//Request var
	eRequestedProfile		: E_AXIS_MOVE_PROFILE := E_AXIS_MOVE_PROFILE.Slow;
	rRequestedTarget		: LREAL := 0;
	Profile				    	: ARRAY[0..2]OF ST_AXIS_MOVE_PROFILE ;
END_VAR

IF NOT bInit THEN
  RETURN;
END_IF

//CALL BLOCK
fbPower(Axis:= _AxisREF_P^, Override:= lrAxisOverride);
fbStop(Axis:= _AxisREF_P^);
fbReset(Axis:= _AxisREF_P^);
fbHome( Axis:= _AxisREF_P^, bCalibrationCam:=_udCalibrationSensor_P^.19,
		    Options := stHomingOption, Position := lrnOffsetExtractorHoming);
fbHomeInv( Axis:= _AxisREF_P^, bCalibrationCam:=_udCalibrationSensor_P^.19,
		    Options := stHomingInvOption, Position := lrnOffsetExtractorHoming);
fbMoveAbso(Axis:= _AxisREF_P^);
fbReadStatus(Axis:= _AxisREF_P^,Enable := TRUE);
fbMoveJog(Axis := _AxisREF_P^,JogForward := stJogControl.bMoveFW, JogBackwards := stJogControl.bMoveBW);
fbTimeRetryHomming(IN := nStep = E_StepAxis.AbortHoming);
fbTimeAbortHoming(IN := nStep = E_StepAxis.RetryHoming);
fbTimeOutReset(IN := nStep = E_StepAxis.InitReset);
fbTrigErrorMotor(CLK := _AxisREF_P^.NcToPlc.ErrorCode <> 0);
_lrActPos := _AxisREF_P^.NcToPlc.ActPos;


IF fbTrigErrorMotor.Q THEN
  nStep := E_StepAxis.Idle;
  bRequestMoveAbso := FALSE;
  bRequestHoming := FALSE;
  fbHome.Execute := FALSE;
  fbHomeInv.Execute := FALSE;
  fbMoveAbso.Execute := FALSE;
END_IF

//Defect
objMotorError();
objMotorError.Set(bSetActivate := _AxisREF_P^.NcToPlc.ErrorCode <> 0 AND _AxisREF_P^.NcToPlc.ErrorCode <> 18000 );

objMoveAbsError();
objMoveAbsError.Set(bSetActivate := fbMoveAbso.Error AND fbMoveAbso.Execute);

objMotorResetError();
objMotorResetError.Set(bSetActivate := fbReset.Error AND fbReset.Execute);

//objMotorPowerError();
//objMotorPowerError.SetState(bSetActivate := fbPower.Error AND fbPower.Enable);

objHommingError();

// If bEnableMove is down, do a stop automatically
//IF NOT bEnableMove THEN
//	bRequestStop		:= TRUE;
//	eRequestedProfile	:= E_AXIS_MOVE_PROFILE.Fast;
//END_IF


CASE nStep OF
	// ------------------------------------------------------------------
	E_StepAxis.IDLE :	
		bRequestStop	:= FALSE;			
    IF bRequestPowerOff THEN
      nStep := E_StepAxis.PoweringOff;
      bRequestPowerOff	:= FALSE;
    ELSIF bRequestPowerOn THEN
      nStep := E_StepAxis.PoweringOn;
      bRequestPowerOn		:= FALSE;
    ELSIF bRequestMoveAbso THEN
      nStep := E_StepAxis.InitMoveAbs;
      bRequestMoveAbso	:= FALSE;
    ELSIF bRequestHoming THEN
      bRequestHoming		:= FALSE;
			IF _udCalibrationSensor_P^.19 THEN
				nStep := E_StepAxis.InitRetryHoming;
			ELSE
				nStep := E_StepAxis.InitHoming;
			END_IF	
    ELSIF bRequestReset OR (_AxisREF_P^.NcToPlc.ErrorCode <> 0) THEN
			//added to support MDF extractor: homing in both direction		
			nStep := E_StepAxis.InitReset;
      bRequestReset		:= FALSE;
    END_IF
	
	// ******************************************************************
	// --- POWER ---
	// ******************************************************************
		// ------------------------------------------------------------------
		E_StepAxis.PoweringOff :
      fbPower.Enable := FALSE;
			objHommingError.Set(Activate:= FALSE);
      IF NOT fbPower.Status THEN
        _bIsDone	:= TRUE;
        _bIsBusy	:= FALSE;
        nStep := E_StepAxis.IDLE;
      ELSIF fbPower.Error THEN
        nErrorId := fbPower.ErrorID;
        nStep := E_StepAxis.ERROR;
      END_IF
			
		// ------------------------------------------------------------------
		E_StepAxis.PoweringOn :
      fbPower.Enable			:= TRUE;
      fbPower.Enable_Positive	:= TRUE;
      fbPower.Enable_Negative	:= TRUE;
      IF fbPower.Status THEN
        _bIsDone	:= TRUE;
        _bIsBusy	:= FALSE;
        nStep  := E_StepAxis.Idle;
      ELSIF fbPower.Error THEN
        fbPower.Enable			:= FALSE;
        fbPower.Enable_Positive	:= FALSE;
        fbPower.Enable_Negative	:= FALSE;
        _bIsBusy	:= FALSE;
        nStep  := E_StepAxis.Idle;      
      END_IF
			
	// ******************************************************************
	// --- ABSOLUTE ---
	// ******************************************************************
		// ------------------------------------------------------------------
		E_StepAxis.InitMoveAbs:
      fbMoveAbso.Position		:= rRequestedTarget;
      fbMoveAbso.Velocity		:= Profile[eRequestedProfile].Velo;
      fbMoveAbso.Acceleration	:= Profile[eRequestedProfile].Acc;
      fbMoveAbso.Deceleration	:= Profile[eRequestedProfile].Dec;
      fbMoveAbso.Jerk			:= Profile[eRequestedProfile].Jerk;
      fbMoveAbso.Execute			:= TRUE;
      IF fbMoveAbso.Busy THEN
         nStep := E_StepAxis.MoveAbs;
      END_IF
    
    // ------------------------------------------------------------------  
    E_StepAxis.MoveAbs:    
      IF fbMoveAbso.Done THEN
        nStep:= E_StepAxis.EndMoveAbs;
      ELSIF bRequestStop THEN
        fbMoveAbso.Execute := FALSE;
        nStep:= E_StepAxis.InitStop;
        bRequestStop := FALSE;
      ELSIF fbMoveAbso.Error THEN
        fbMoveAbso.Execute	:= false;
        _bIsBusy	:= FALSE;
        nStep     := E_StepAxis.Idle;
      END_IF
     
    // ------------------------------------------------------------------  
    E_StepAxis.EndMoveAbs: 
      _bIsDone	:= TRUE;
      _bIsBusy	:= FALSE;
      fbMoveAbso.Execute  := FALSE;
      nStep     := E_StepAxis.Idle;
						
	// ******************************************************************
	// --- STOP ---
	// ******************************************************************
		// ------------------------------------------------------------------
		E_StepAxis.InitStop :
			bRequestStop	:= FALSE;
      fbStop.Deceleration	:= Profile[eRequestedProfile].Dec;
      fbStop.Jerk			    := Profile[eRequestedProfile].Jerk;
      fbStop.Execute		  := TRUE;
      IF fbStop.Busy THEN
        nStep := E_StepAxis.Stopping;
			END_IF
                  
		// ------------------------------------------------------------------
		E_StepAxis.Stopping :        
      IF _AxisREF_P^.Status.NotMoving THEN
        _bIsDone	:= TRUE;
        _bIsBusy	:= FALSE;
        nStep  := E_StepAxis.EndStopping;
      END_IF
        
		// ------------------------------------------------------------------
		E_StepAxis.EndStopping :        
      fbStop.Execute	:= FALSE;
      objHommingError.Set(Activate:= FALSE);
			nStep           := E_StepAxis.Idle;

	// ******************************************************************
	// --- HOMING ---
	// ******************************************************************
		// ------------------------------------------------------------------
		E_StepAxis.InitHoming:
      fbHome.Execute			:= TRUE;
      IF fbHome.Busy THEN
        nStep := E_StepAxis.Homing;
			END_IF      
    
    // ------------------------------------------------------------------  
    E_StepAxis.Homing:    
      IF fbHome.Done THEN
        nStep:= E_StepAxis.EndHoming;
      ELSIF bRequestStop THEN
        fbHome.Execute			:= false;
        nStep:= E_StepAxis.InitStop;
        bRequestStop := FALSE;
      ELSIF _nAxisTorque_P^ < -800  THEN
        nStep:= E_StepAxis.InitAbortHoming;    
      END_IF
 
		// ------------------------------------------------------------------
		E_StepAxis.InitAbortHoming:
      fbStop.Deceleration	:= Profile[eRequestedProfile].Dec;
      fbStop.Jerk			    := Profile[eRequestedProfile].Jerk;
      fbStop.Execute		  := TRUE;
      fbHome.Execute			:= FALSE;
      IF fbStop.Busy THEN
        nStep := E_StepAxis.AbortHoming;
			END_IF
      
		// ------------------------------------------------------------------
		E_StepAxis.AbortHoming:
      IF _AxisREF_P^.Status.NotMoving AND fbTimeRetryHomming.Q THEN
        fbStop.Execute	:= FALSE;
        nStep  := E_StepAxis.InitRetryHoming;
      END_IF    
    
    // ------------------------------------------------------------------  
    E_StepAxis.EndHoming: 
      _bIsDone	:= TRUE;
      _bIsBusy	:= FALSE;
      fbHome.Execute			:= FALSE;
      fbHomeInv.Execute			:= FALSE;
      nStep                   := E_StepAxis.Idle;
    
    // ------------------------------------------------------------------   
		E_StepAxis.InitRetryHoming:
      fbHomeInv.Execute			:= TRUE;
      IF fbHomeInv.Busy THEN
        lrSetHomingCheckPos := _AxisREF_P^.NcToPlc.ActPos;
        nStep := E_StepAxis.RetryHoming;
			END_IF  

    // ------------------------------------------------------------------  
    E_StepAxis.RetryHoming:    
      IF fbHomeInv.Done THEN
        nStep:= E_StepAxis.EndHoming;
      ELSIF bRequestStop THEN
        fbHomeInv.Execute			:= FALSE;
        nStep:= E_StepAxis.InitStop;
        bRequestStop := FALSE;
      ELSIF  (_nAxisTorque_P^ > 600) THEN
        nStep:= E_StepAxis.InitStop;
        fbHomeInv.Execute := FALSE;
        objHommingError.Set(Activate:= TRUE);      
      END_IF
			
	// ******************************************************************
	// --- RESETTING ---
	// ******************************************************************
  	// ------------------------------------------------------------------
		E_StepAxis.InitReset :
      fbReset.Execute		:= TRUE;
      IF fbTimeOutReset.Q THEN
        nStep := E_StepAxis.EndReset;
			END_IF
      IF fbReset.Busy THEN
        nStep := E_StepAxis.Resetting;
      END_IF
      
    // ------------------------------------------------------------------
		E_StepAxis.Resetting :
      IF fbReset.Done THEN
        bError	:= FALSE;
        _bIsDone	:= TRUE;
        _bIsBusy	:= FALSE;
        nStep := E_StepAxis.EndReset;
      END_IF
      
		// ------------------------------------------------------------------
		E_StepAxis.EndReset:
      fbReset.Execute	:= FALSE;
      nStep := E_StepAxis.Idle;
			
	// ******************************************************************
	// --- ERROR ---
	// ******************************************************************
		// ------------------------------------------------------------------
		E_StepAxis.ERROR :
				//added by Tristan 23-4-2024
				fbPower.Enable			:= FALSE;
        fbPower.Enable_Positive	:= FALSE;
        fbPower.Enable_Negative	:= FALSE;
				      fbHome.Execute			:= FALSE;
      fbHomeInv.Execute			:= FALSE;
			bRequestStop := FALSE;
      bError	:= TRUE;
      _bIsBusy	:= FALSE;
END_CASE

// Call again to refresh cmd
fbPower(Axis:= _AxisREF_P^, Override:= lrAxisOverride);
fbStop(Axis:= _AxisREF_P^);
fbReset(Axis:= _AxisREF_P^);
fbHome( Axis:= _AxisREF_P^, bCalibrationCam:=_udCalibrationSensor_P^.19,
		    Options := stHomingOption, Position := lrnOffsetExtractorHoming);
fbHomeInv( Axis:= _AxisREF_P^, bCalibrationCam:=_udCalibrationSensor_P^.19,
		    Options := stHomingInvOption, Position := lrnOffsetExtractorHoming);
fbMoveAbso(Axis:= _AxisREF_P^);
fbReadStatus(Axis:= _AxisREF_P^,Enable := TRUE);

Case01Hysto( nStep);

PROPERTY bIsBusy : bool
GET
bIsBusy := _bIsBusy;
END_GET
END_PROPERTY

PROPERTY bIsDone : bool
GET
bIsDone := _bIsDone;
END_GET
END_PROPERTY

PROPERTY bIsHomed : bool
GET
IF _AxisREF_P <> 0 THEN
	bIsHomed := _AxisREF_P^.Status.Homed;
END_IF
END_GET
END_PROPERTY

PROPERTY bIsInPos : bool
GET
bIsInPos := _AxisREF_P^.Status.InPositionArea;
END_GET
END_PROPERTY

PROPERTY bIsPowered : bool
GET
bIsPowered :=  fbPower.Status;
END_GET
END_PROPERTY

PROPERTY bIsStopped : BOOL
GET
bIsStopped := _AxisREF_P^.Status.NotMoving;
END_GET
END_PROPERTY

PROPERTY InError : bool
GET
InError := _AxisREF_P^.NcToPlc.ErrorCode <> 0;
END_GET
END_PROPERTY

METHOD Init : BOOL
VAR_INPUT
	AxisREF_P				      	: POINTER TO AXIS_REF;
  bHomingSensor_P			    : POINTER TO BOOL;
  nAxisTorque_P           : POINTER TO INT;
  nLineNumber_P           : POINTER TO INT;
END_VAR

// Class ID: 201
IF NOT bInit and nAxisTorque_P <> 0 AND bHomingSensor_P <> 0 AND nLineNumber_P <> 0 AND AxisREF_P <> 0 THEN
  bInit := TRUE;

	_udCalibrationSensor_P := bHomingSensor_P;
	_AxisREF_P := AxisREF_P;
	_LineNumber_P := nLineNumber_P;
	_nAxisTorque_P :=  nAxisTorque_P;
	
	stHomingOption.SearchDirection := MC_Direction.MC_Negative_Direction;
	stHomingOption.SyncDirection := MC_Direction.MC_Positive_Direction;
	stHomingInvOption.SearchDirection := MC_Direction.MC_Positive_Direction;
	stHomingInvOption.SyncDirection := MC_Direction.MC_Positive_Direction;
	
//	// Defect
//	objMotorError.Register(GVL.objDefectManager,CidCL.sClassID_Axis_C[(nLineNumber_P^)+C.usiNbAxisOutSpan_C],CidErr.sErrorIDs_Axis_C[1]);
//	objMoveAbsError.Register(GVL.objDefectManager,CidCL.sClassID_Axis_C[(nLineNumber_P^)+C.usiNbAxisOutSpan_C],CidErr.sErrorIDs_Axis_C[2]);
//	objMotorResetError.Register(GVL.objDefectManager,CidCL.sClassID_Axis_C[(nLineNumber_P^)+C.usiNbAxisOutSpan_C],CidErr.sErrorIDs_Axis_C[3]);
//	objMotorPowerError.Register(GVL.objDefectManager,CidCL.sClassID_Axis_C[(nLineNumber_P^)+C.usiNbAxisOutSpan_C],CidErr.sErrorIDs_Axis_C[4]);
//	objHommingError.Register(GVL.objDefectManager,CidCL.sClassID_Axis_C[(nLineNumber_P^)+C.usiNbAxisOutSpan_C],CidErr.sErrorIDs_Axis_C[5]);
	// CAUTION: not possible to indicate the line by this way
  // => Future fix: use the location Infos in the database (maybe by using another stored procedure)
	InitDefect(iNumInst := nLineNumber_P^);
END_IF
END_METHOD

METHOD PRIVATE InitDefect : BOOL
VAR_INPUT
	iNumInst	:	INT;
END_VAR
	// Defect
//	objMotorError.Register(GVL.objDefectManager,CidCL.sClassID_Axis_C[iNumInst+C.usiNbAxisOutSpan_C],CidErr.sErrorIDs_Axis_C[1]);
//	objMoveAbsError.Register(GVL.objDefectManager,CidCL.sClassID_Axis_C[iNumInst+C.usiNbAxisOutSpan_C],CidErr.sErrorIDs_Axis_C[2]);
//	objMotorResetError.Register(GVL.objDefectManager,CidCL.sClassID_Axis_C[iNumInst+C.usiNbAxisOutSpan_C],CidErr.sErrorIDs_Axis_C[3]);
//	objMotorPowerError.Register(GVL.objDefectManager,CidCL.sClassID_Axis_C[iNumInst+C.usiNbAxisOutSpan_C],CidErr.sErrorIDs_Axis_C[4]);
//	objHommingError.Register(GVL.objDefectManager,CidCL.sClassID_Axis_C[iNumInst+C.usiNbAxisOutSpan_C],CidErr.sErrorIDs_Axis_C[5]);

	objMotorError.Register(GVL.objDefectManager,CidCL.sClassID_Axis_C[iNumInst+C.usiNbAxisOutSpan_C],CidErr.sAxisGeneralErrorMC);
	objMoveAbsError.Register(GVL.objDefectManager,CidCL.sClassID_Axis_C[iNumInst+C.usiNbAxisOutSpan_C],CidErr.sAxisMovingErrorMC);
	objMotorResetError.Register(GVL.objDefectManager,CidCL.sClassID_Axis_C[iNumInst+C.usiNbAxisOutSpan_C],CidErr.sAxisResetErrorMC);
	objMotorPowerError.Register(GVL.objDefectManager,CidCL.sClassID_Axis_C[iNumInst+C.usiNbAxisOutSpan_C],CidErr.sAxisPowerErrorMC);
	objHommingError.Register(GVL.objDefectManager,CidCL.sClassID_Axis_C[iNumInst+C.usiNbAxisOutSpan_C],CidErr.sAxisHomingOutBound);
	
	(*	Proposition for the database: clear separation between fixed and variable number of objects across the installation
	objMotorError.Register(GVL.objDefectManager,CidCL.sClassID_Axis_C[iNumInst],CidErr.sAxisGeneralErrorMC);
	objMoveAbsError.Register(GVL.objDefectManager,CidCL.sClassID_Axis_C[iNumInst],CidErr.sAxisMovingErrorMC);
	objMotorResetError.Register(GVL.objDefectManager,CidCL.sClassID_Axis_C[iNumInst],CidErr.sAxisResetErrorMC);
	objMotorPowerError.Register(GVL.objDefectManager,CidCL.sClassID_Axis_C[iNumInst],CidErr.sAxisPowerErrorMC);
	objHommingError.Register(GVL.objDefectManager,CidCL.sClassID_Axis_C[iNumInst],CidErr.sAxisHomingOutBound);
	
*)
END_METHOD

PROPERTY lrActPos : lreal
GET
lrActPos := _lrActPos;
END_GET
END_PROPERTY

PROPERTY lrActTorque : lreal
GET
lrActTorque := _AxisREF_P^.NcToPlc.ActTorque;
END_GET
END_PROPERTY

{attribute 'TcRpcEnable'}
METHOD RequestHoming : bool
VAR_INPUT
	lrnOffsetExtractorHomingRef : LREAL;
END_VAR
_bIsDone			:= FALSE;
IF bIsPowered AND bEnableMove AND NOT bError THEN
	bRequestHoming 		:= TRUE;
	_bIsBusy				    := TRUE;
	lrnOffsetExtractorHoming := lrnOffsetExtractorHomingRef;
END_IF
END_METHOD

{attribute 'TcRpcEnable'}
METHOD RequestMove : BOOL
VAR_INPUT
	Profile	: E_AXIS_MOVE_PROFILE;
	Target	: LREAL;
END_VAR
_bIsDone		:= FALSE;

IF bIsPowered AND bEnableMove AND NOT bError AND NOT bIsBusy THEN
  _bIsBusy				  := TRUE;
  bRequestMoveAbso	:= TRUE;
  eRequestedProfile	:= Profile;
  rRequestedTarget	:= Target;
END_IF
END_METHOD

{attribute 'TcRpcEnable'}
METHOD RequestPowerOFF : BOOL
VAR_INPUT
END_VAR
_bIsDone			:= FALSE;

IF bIsPowered AND NOT bIsBusy THEN
	bRequestPowerOFF	:= TRUE;
	_bIsBusy				:= TRUE;
END_IF
END_METHOD

{attribute 'TcRpcEnable'}
METHOD RequestPowerON : bool
VAR_INPUT
END_VAR
_bIsDone			:= FALSE;

IF NOT bIsPowered AND NOT bError THEN
	bRequestPowerON		:= TRUE;
	_bIsBusy				  := TRUE;
END_IF
END_METHOD

{attribute 'TcRpcEnable'}
METHOD RequestReset :bool
VAR_INPUT
END_VAR
_bIsDone			:= FALSE;

IF TRUE(*bError*) THEN
	bRequestReset 		:= TRUE;
	_bIsBusy				:= TRUE;
	nErrorId			:= 0;
END_IF
END_METHOD

{attribute 'TcRpcEnable'}
METHOD RequestStop : bool
VAR_INPUT
	Profile	: E_AXIS_MOVE_PROFILE;
END_VAR
_bIsDone		:= FALSE;
IF _bIsBusy THEN
  _bIsBusy := false;
	bRequestStop := TRUE;
	eRequestedProfile	:= Profile;
END_IF
END_METHOD

{attribute 'TcRpcEnable'}
METHOD SetAxisProfile : BOOL
VAR_INPUT
	Profile			: E_AXIS_MOVE_PROFILE;
	Velocity		: REAL;
	Acceleration	: REAL;
	Deceleration	: REAL;
	Jerk			: REAL;
END_VAR
THIS^.Profile[Profile].Velo		:= Velocity;
THIS^.Profile[Profile].Acc		:= Acceleration;
THIS^.Profile[Profile].Dec		:= Deceleration;
THIS^.Profile[Profile].Jerk		:= Jerk;
END_METHOD

END_FUNCTION_BLOCK

// ---- POUs/FB_testAxleAllJog.TcPOU
FUNCTION_BLOCK FB_testAxleAllJog 
VAR
 	stm	: UINT := 10;
  stIRL : ST_LineReference;
  bFW, bBW, b : BOOL := FALSE;
END_VAR

G.AxisL1LeftFront(); 
G.AxisL2RightFront();
G.AxisL1LeftBack();
G.AxisL2RightBack();
G.AxisMaster();

CASE stm OF   
  10:
    stIRL.nThis := 0;
    stIRL.nFixedID := 1;
    b := G.AxisL1LeftFront.Init(stIrrLine := stIRL, stAxisMotor_P := ADR(G.stAX.L1LeftFront), stAxisMaster_P := ADR(G.stAX.Master));
    b := b and G.AxisL2RightFront.Init(stIrrLine := stIRL, stAxisMotor_P := ADR(G.stAX.L2RightFront), stAxisMaster_P := ADR(G.stAX.Master));
    b := b and G.AxisL1LeftBack.Init(stIrrLine := stIRL, stAxisMotor_P := ADR(G.stAX.L1LeftBack), stAxisMaster_P := ADR(G.stAX.Master));
    b := b and G.AxisL2RightBack.Init(stIrrLine := stIRL, stAxisMotor_P := ADR(G.stAX.L2RightBack), stAxisMaster_P := ADR(G.stAX.Master));
    b := b and G.AxisMaster.Init(stIrrLine := stIRL, stAxisMotor_P := ADR(G.stAX.Master), stAxisMaster_P := ADR(G.stAX.Master));
    if b then
      stm := 1000;
		END_IF   
 
  1000:
    IF NOT G.AxisL1LeftFront.IsBusy AND NOT G.AxisL2RightFront.IsBusy AND NOT G.AxisL1LeftBack.IsBusy AND NOT G.AxisL2RightBack.IsBusy AND NOT G.AxisMaster.IsBusy THEN
      G.AxisL1LeftFront.RequPowerOn();
      G.AxisL2RightFront.RequPowerOn();
      G.AxisL1LeftBack.RequPowerOn();
      G.AxisL2RightBack.RequPowerOn();
      //G.AxisMaster.RequPowerOn();
      stm := 1120;
    END_IF
    
  1120:
    IF G.AxisL1LeftFront.IsDone AND G.AxisL2RightFront.IsDone AND G.AxisL1LeftBack.IsDone AND G.AxisL2RightBack.IsDone THEN //AND G.AxisMaster.IsDone
      stm := 1130;
    END_IF
    
  1130:
    IF NOT G.AxisL1LeftFront.IsError AND NOT G.AxisL2RightFront.IsError AND NOT G.AxisL1LeftBack.IsError AND NOT G.AxisL2RightBack.IsError THEN // AND NOT G.AxisMaster.IsError 
      stm := 1140;
    ELSE
      stm := 0;
    END_IF
  
  1140:
    IF G.AxisL1LeftFront.IsDone AND G.AxisL2RightFront.IsDone AND G.AxisL1LeftBack.IsDone AND G.AxisL2RightBack.IsDone THEN //AND G.AxisMaster.IsDone
      stm := 1150;
    END_IF
    
  1150:
    IF NOT G.AxisL1LeftFront.IsError AND NOT G.AxisL2RightFront.IsError AND NOT G.AxisL1LeftBack.IsError AND NOT G.AxisL2RightBack.IsError THEN // AND NOT G.AxisMaster.IsError 
      stm := 2000;
    ELSE
      stm := 0;
    END_IF
  
  2000:
    bFW := true;
    bBW := FALSE;
    G.AxisL1LeftFront.JogExec(bExecIn := TRUE, bExecJogFWIn := bFW, bExecJogBWIn := bBW);
    G.AxisL1LeftBack.JogExec(bExecIn := TRUE, bExecJogFWIn := bFW, bExecJogBWIn := bBW);
    G.AxisL2RightFront.JogExec(bExecIn := TRUE, bExecJogFWIn := bFW, bExecJogBWIn := bBW);
    G.AxisL2RightBack.JogExec(bExecIn := TRUE, bExecJogFWIn := bFW, bExecJogBWIn := bBW);
    stm := 2000;
  
  0:; //park 
END_CASE

(*
  140:
    IF NOT G.AxisL1LeftFront.IsBusy THEN
      G.AxisL1LeftFront.RequGearInDyn();
      stm := 150;
    END_IF
  150:
    IF G.AxisL1LeftFront.IsDone THEN
      stm := 160;
    END_IF
  160:
    IF NOT G.AxisL1LeftFront.IsError THEN
      stm := 170; 
    ELSE
      stm := 0;
    END_IF
    
  170:
    IF NOT G.AxisMaster.IsBusy THEN
      G.AxisMaster.RequJogAxisMaster();
      stm := 180;
    END_IF
    
  2000:
    bFW := FALSE;
    bBW := FALSE;
    G.AxisMaster.JogExec(bExecIn := TRUE, bExecJogFWIn := bFW, bExecJogBWIn := bBW);
    stm := 180;
*)

END_FUNCTION_BLOCK

// ---- POUs/FB_PowerAxis1.TcPOU
FUNCTION_BLOCK FB_PowerAxis1
VAR
  stm	: UINT := 10;
  bFW, bBW,bPower,bReset,bResetDone,bError,bBusy,bPowerStatus : BOOL := FALSE;
  errId : UDINT;
  
  fbPower : MC_Power;
  fbReset : MC_Reset;
END_VAR

fbPower(
	Axis:= G.stAX.L1LeftFront, 
	Enable:= bPower, 
	Enable_Positive:= bPower, 
	Enable_Negative:= bPower, 
	Override:= 100.0, 
  Status=>bPowerStatus,
	Busy=>bBusy , 
	Error=>bError, 
	ErrorID=> errId);

fbReset(
	Axis:= G.stAX.L1LeftFront, 
	Execute:= bReset, 
	Done=> bResetDone,
	Busy=> bBusy, 
	Error=>bError, 
	ErrorID=>errId);
  
CASE stm OF 
  10:
		bPower := TRUE;
		stm := 20;
	20:
		IF G.stAX.L1LeftFront.Status.Error THEN //really at the level of NC
			stm := 30;
		ELSE
			stm := 50;
		END_IF
	30:
		bReset := TRUE;
		stm := 40;	
	40:
		IF bResetDone THEN
			bReset := FALSE;
			stm := 50;
		END_IF
	50:
    bPowerStatus := fbPower.Status;
		IF bPowerStatus THEN
			stm := 0;
		END_IF
   
  0:stm := 0;
END_CASE

END_FUNCTION_BLOCK

// ---- POUs/FB_PowerMaster.TcPOU
FUNCTION_BLOCK FB_PowerMaster
VAR
  stm	: UINT := 10;
  bFW, bBW,bPower,bReset,bResetDone,bError,bBusy,bPowerStatus : BOOL := FALSE;
  errId : UDINT;
  
  fbPower : MC_Power;
  fbReset : MC_Reset;
END_VAR

fbPower(
	Axis:= G.stAX.Master, 
	Enable:= bPower, 
	Enable_Positive:= bPower, 
	Enable_Negative:= bPower, 
	Override:= 100.0, 
  Status=>bPowerStatus,
	Busy=>bBusy , 
	Error=>bError, 
	ErrorID=> errId);

fbReset(
	Axis:= G.stAX.Master, 
	Execute:= bReset, 
	Done=> bResetDone,
	Busy=> bBusy, 
	Error=>bError, 
	ErrorID=>errId);
  
CASE stm OF 
  10:
		bPower := TRUE;
 		stm := 20;
	20:
		IF G.stAX.Master.Status.Error THEN //really at the level of NC
			stm := 30;
		ELSE
			stm := 50;
		END_IF
	30:
		bReset := TRUE;
		stm := 40;	
	40:
		IF bResetDone THEN
			bReset := FALSE;
			stm := 50;
		END_IF
	50:
    bPowerStatus := fbPower.Status;
		IF bPowerStatus THEN
			stm := 0;
		END_IF
   
  0:stm := 0;
END_CASE

END_FUNCTION_BLOCK

// ---- POUs/FB_testAxisL1LeftFrontJog.TcPOU
FUNCTION_BLOCK FB_testAxisL1LeftFrontJog 
VAR
 	stm	: UINT := 10;
  stIRL : ST_LineReference;
  b, bFW, bBW : BOOL := FALSE;
END_VAR

G.AxisL1LeftFront(); 
//G.AxisL2RightFront();
//G.AxisL1LeftBack();
//G.AxisL2RightBack();
//G.AxisMaster();

CASE stm OF   
  10:
    stIRL.nThis := 0;
    stIRL.nFixedID := 1;
    b := G.AxisL1LeftFront.Init(stIrrLine := stIRL, stAxisMotor_P := ADR(G.stAX.L1LeftFront), stAxisMaster_P := ADR(G.stAX.Master));
    //G.AxisL2RightFront.Init(stIrrLine := stIRL, stAxisMotor_P := ADR(G.stAX.L2RightFront), stAxisMaster_P := ADR(G.stAX.Master));
    //G.AxisL1LeftBack.Init(stIrrLine := stIRL, stAxisMotor_P := ADR(G.stAX.L1LeftBack), stAxisMaster_P := ADR(G.stAX.Master));
    //G.AxisL2RightBack.Init(stIrrLine := stIRL, stAxisMotor_P := ADR(G.stAX.L2RightBack), stAxisMaster_P := ADR(G.stAX.Master));
    //G.AxisMaster.Init(stIrrLine := stIRL, stAxisMotor_P := ADR(G.stAX.Master), stAxisMaster_P := ADR(G.stAX.Master));
    if b then
      stm := 50;
		END_IF   

  50:
    IF NOT G.AxisL1LeftFront.IsBusy THEN
      G.AxisL1LeftFront.RequPowerOn();
      stm := 60;
    END_IF
  60:
    IF G.AxisL1LeftFront.IsDone THEN
      stm := 70;
    END_IF
  70:
    IF NOT G.AxisL1LeftFront.IsError THEN
      stm := 100;
    ELSE
      stm := 0;
    END_IF

  100:
    IF NOT G.AxisL1LeftFront.IsBusy THEN
      G.AxisL1LeftFront.RequJogAxisMaster();
      bFW := true;
      stm := 110;
    END_IF

  110:
    IF G.AxisL1LeftFront.IsDone THEN
      stm := 120;
    END_IF
    
  120:
    IF NOT G.AxisL1LeftFront.IsError THEN
      stm := 130;
    ELSE
      stm := 0;
    END_IF

  130:
    bFW := true;
    bBW := FALSE;
    G.AxisL1LeftFront.JogExec(bExecIn := TRUE, bExecJogFWIn := bFW, bExecJogBWIn := bBW);
    stm := 130;
  
  0:; //park 
END_CASE

END_FUNCTION_BLOCK

// ---- POUs/AxisDay2Training/FB_AxisStMachine.TcPOU
FUNCTION_BLOCK FB_AxisStMachine
VAR_IN_OUT
	AxisInOut : AXIS_REF;//AXIS_REF contains input and output
END_VAR
VAR
	nStep : UINT := 10;
	
	fbPower : MC_Power;
		
	errId : UDINT;
	bBusy, bError, bMoveAbs, bMoveVel, bDone, bPower, bReset, bResetDone,bVelocity, bInVelocity, MoveAbsbDone, bDoneHalt, bAborted,bHalt,bHomingDone : BOOL;

	bDemandStop,bDemandVel  AT%I* : BOOL;
	
	fbMoveAbs : MC_MoveAbsolute;
	fTarget	: LREAL := 720;
	fVelocity : LREAL := 36;
	fVelocityInfinite : LREAL := 360;
	fbReset : MC_Reset;//remove error in the NC only for AX8000 but not for AX5000
	fbVelocity : MC_MoveVelocity;
	fbHalt : MC_HALT;
	fbHome : MC_Home;
	bCalibCam AT%I* : BOOL;
	bHome : BOOL;
END_VAR

RunFBs();

CASE nStep OF
	0 : //Idle
		;
	10:
		bPower := TRUE;
		nStep := 15;
	15:
		IF AxisInOut.Status.Error THEN //really at the level of NC
			nStep := 20;
		ELSE
			nstep := 40;
		END_IF
	20:
		bReset := TRUE;
		nstep := 30;	
	30:
		IF bResetDone THEN
			bReset := FALSE;
			nStep := 40;
		END_IF
	40:
		IF fbPower.Status THEN
			bHome := TRUE;
			nStep := 45;
		END_IF
	45:
		IF bHomingDone THEN
			bHome := FALSE;
			nStep := 50;
		END_IF 
	50:
		bMoveAbs := TRUE;
		fTarget	 := 36;//gradi
		fVelocity := 36;
		nstep := 60;
	60:
		IF MoveAbsbDone THEN
			bMoveAbs := FALSE;
			nStep := 65;
		END_IF
	65:
		IF bDemandVel THEN
			nStep := 70;
		END_IF
	70:
		bMoveVel := TRUE;
		fVelocityInfinite := 1440;
		nStep := 80;
	80:
		IF bDemandStop THEN
			bMoveVel := FALSE;
			nStep := 90;
		END_IF
	90:
		bHalt := TRUE;
		nStep := 100;
	
	100:
		IF fbHalt.Done THEN
			bHalt := FALSE;
			nStep := 0;
		END_IF
	ELSE
		;
END_CASE

METHOD RunFBs : BOOL
fbPower(
	Axis:= AxisInOut, 
	Enable:= bPower, 
	Enable_Positive:= TRUE, 
	Enable_Negative:= TRUE, 
	Override:= 100, 
	Busy=>bBusy , 
	Error=>bError, 
	ErrorID=> errId);

fbMoveAbs(
	Axis:= AxisInOut, 
	Execute:= bMoveAbs, 
	Position:= fTarget, 
	Velocity:= fVelocity,  
	Done=> MoveAbsbDone, 
	Busy=>bBusy, 
	Error=>bError, 
	ErrorID=> errId);

fbReset(
	Axis:= AxisInOut, 
	Execute:= bReset, 
	Done=> bResetDone,
	Busy=> bBusy, 
	Error=>bError, 
	ErrorID=>errId);
	
fbVelocity(
	Axis:= AxisInOut, 
	Execute:= bMoveVel, 
	Velocity:= fVelocityInfinite, 
	InVelocity=> bInVelocity, 
	Busy=> bBusy, 
	Error=>bError, 
	ErrorID=>errId);

fbHalt(
	Axis:= AxisInOut, 
	Execute:= bHalt, 
	Done=> bDoneHalt, 
	Busy=> bBusy, 
	CommandAborted=> bAborted, 
	Error=> bError, 
	ErrorID=>errId);

	//without giving special values to the parameters NC parameters are used
fbHome(
	Axis:= AxisInOut, 
	Execute:= bHome, 
	Position:= , 
	HomingMode:= , 
	BufferMode:= , 
	Options:= , 
	bCalibrationCam:= bCalibCam, 
	Done=> bHomingDone, 
	Busy=> , 
	Active=> , 
	CommandAborted=> , 
	Error=> , 
	ErrorID=> );
END_METHOD

END_FUNCTION_BLOCK

// ---- POUs/AxisDay2Training/FB_AxisStMachineMaster.TcPOU
FUNCTION_BLOCK FB_AxisStMachineMaster
VAR_IN_OUT
	AxisInOut : AXIS_REF;//AXIS_REF contains input and output
END_VAR
VAR
	nStep : UINT := 10;
	
	fbPower : MC_Power;
		
	errId : UDINT;
	bBusy, bError, bMoveAbs, bMoveVel, bDone, bPower, bReset, bResetDone,bVelocity, bInVelocity, MoveAbsbDone, bDoneHalt, bAborted,bHalt,bHomingDone : BOOL;

	bDemandStop,bDemandVel  AT%I* : BOOL;
	
	fbMoveAbs : MC_MoveAbsolute;
	fTarget	: LREAL := 720;
	fVelocity : LREAL := 36;
	fVelocityInfinite : LREAL := 360;
	fbReset : MC_Reset;//remove error in the NC only for AX8000 but not for AX5000
	fbVelocity : MC_MoveVelocity;
	fbHalt : MC_HALT;
	fbHome : MC_Home;
	bCalibCam AT%I* : BOOL;
	bHome : BOOL;
END_VAR

RunFBs();

CASE nStep OF
	0 : //Idle
		;
	10:
		bPower := TRUE;
		nStep := 15;
	15:
		IF AxisInOut.Status.Error THEN //really at the level of NC
			nStep := 20;
		ELSE
			nstep := 40;
		END_IF
	20:
		bReset := TRUE;
		nstep := 30;	
	30:
		IF bResetDone THEN
			bReset := FALSE;
			nStep := 40;
		END_IF
	40:
		IF fbPower.Status THEN
			bHome := TRUE;
			nStep := 45;
		END_IF
	45:
		IF bHomingDone THEN
			bHome := FALSE;
			nStep := 50;
		END_IF 
	50:
		bMoveAbs := TRUE;
		fTarget	 := 36;//gradi
		fVelocity := 36;
		nstep := 60;
	60:
		IF MoveAbsbDone THEN
			bMoveAbs := FALSE;
			nStep := 65;
		END_IF
	65:
		IF bDemandVel THEN
			nStep := 70;
		END_IF
	70:
		bMoveVel := TRUE;
		fVelocityInfinite := 1440;
		nStep := 80;
	80:
		IF bDemandStop THEN
			bMoveVel := FALSE;
			nStep := 90;
		END_IF
	90:
		bHalt := TRUE;
		nStep := 100;
	
	100:
		IF fbHalt.Done THEN
			bHalt := FALSE;
			nStep := 0;
		END_IF
	ELSE
		;
END_CASE

METHOD RunFBs : BOOL
fbPower(
	Axis:= AxisInOut, 
	Enable:= bPower, 
	Enable_Positive:= TRUE, 
	Enable_Negative:= TRUE, 
	Override:= 100, 
	Busy=>bBusy , 
	Error=>bError, 
	ErrorID=> errId);

fbMoveAbs(
	Axis:= AxisInOut, 
	Execute:= bMoveAbs, 
	Position:= fTarget, 
	Velocity:= fVelocity,  
	Done=> MoveAbsbDone, 
	Busy=>bBusy, 
	Error=>bError, 
	ErrorID=> errId);

fbReset(
	Axis:= AxisInOut, 
	Execute:= bReset, 
	Done=> bResetDone,
	Busy=> bBusy, 
	Error=>bError, 
	ErrorID=>errId);
	
fbVelocity(
	Axis:= AxisInOut, 
	Execute:= bMoveVel, 
	Velocity:= fVelocityInfinite, 
	InVelocity=> bInVelocity, 
	Busy=> bBusy, 
	Error=>bError, 
	ErrorID=>errId);

fbHalt(
	Axis:= AxisInOut, 
	Execute:= bHalt, 
	Done=> bDoneHalt, 
	Busy=> bBusy, 
	CommandAborted=> bAborted, 
	Error=> bError, 
	ErrorID=>errId);

	//without giving special values to the parameters NC parameters are used
fbHome(
	Axis:= AxisInOut, 
	Execute:= bHome, 
	Position:= , 
	HomingMode:= , 
	BufferMode:= , 
	Options:= , 
	bCalibrationCam:= bCalibCam, 
	Done=> bHomingDone, 
	Busy=> , 
	Active=> , 
	CommandAborted=> , 
	Error=> , 
	ErrorID=> );
END_METHOD

END_FUNCTION_BLOCK
